PROPERTY P_Serial_fbenDTRControl : CtaSysConfig.ITF_BYTE
GET
P_Serial_fbenDTRControl := scParameter.scSerial.fbenDTRControl;
END_GET
END_PROPERTY

PROPERTY P_Serial_fbenParity : CtaSysConfig.ITF_BYTE
GET
P_Serial_fbenParity := scParameter.scSerial.fbenParity;
END_GET
END_PROPERTY

PROPERTY P_Serial_fbenRTSControl : CtaSysConfig.ITF_BYTE
GET
P_Serial_fbenRTSControl := scParameter.scSerial.fbenRTSControl;
END_GET
END_PROPERTY

PROPERTY P_Serial_fbenStopBits : CtaSysConfig.ITF_BYTE
GET
P_Serial_fbenStopBits := scParameter.scSerial.fbenStopBits;
END_GET
END_PROPERTY

PROPERTY P_Serial_fbusiNodeId : CtaSysConfig.ITF_USINT
GET
P_Serial_fbusiNodeId := scParameter.scSerial.fbusiNodeId;
END_GET
END_PROPERTY

PROPERTY P_Serial_fbxEnable : CtaSysConfig.ITF_BOOL
GET
P_Serial_fbxEnable := scParameter.scSerial.fbxEnable;
END_GET
END_PROPERTY

PROPERTY P_Serial_fbxRtuAscii : CtaSysConfig.ITF_BOOL
GET
P_Serial_fbxRtuAscii := scParameter.scSerial.fbxRtuAscii;
END_GET
END_PROPERTY

PROPERTY P_Serial_fbxEnableWatchDog : CtaSysConfig.ITF_BOOL
GET
P_Serial_fbxEnableWatchDog := scParameter.scSerial.fbxEnableWatchDog;
END_GET
END_PROPERTY

PROPERTY P_Serial_fbtWatchDog : CtaSysConfig.ITF_TIME
GET
P_Serial_fbtWatchDog := scParameter.scSerial.fbtWatchDog;
END_GET
END_PROPERTY

PROPERTY P_Serial_fbenPort : CtaSysConfig.ITF_INT
GET
P_Serial_fbenPort := scParameter.scSerial.fbenPort;
END_GET
END_PROPERTY

PROPERTY P_Tcp_fbxEnable : CtaSysConfig.ITF_BOOL
GET
P_Tcp_fbxEnable := scParameter.scTcp.fbxEnable;
END_GET
END_PROPERTY

PROPERTY P_Tcp_fbwPort : CtaSysConfig.ITF_WORD
GET
P_Tcp_fbwPort := scParameter.scTcp.fbwPort;
END_GET
END_PROPERTY

PROPERTY P_Tcp_fbxEnableWatchDog : CtaSysConfig.ITF_BOOL
GET
P_Tcp_fbxEnableWatchDog := scParameter.scTcp.fbxEnableWatchDog;
END_GET
END_PROPERTY

PROPERTY P_Tcp_fbtWatchDog : CtaSysConfig.ITF_TIME
GET
P_Tcp_fbtWatchDog := scParameter.scTcp.fbtWatchDog;
END_GET
END_PROPERTY

PROPERTY P_Tcp_fbstInterface : CtaSysConfig.ITF_STRING40
GET
P_Tcp_fbstInterface := scParameter.scTcp.fbstInterface;
END_GET
END_PROPERTY

END_FUNCTION_BLOCK

// 21 Interface/SERVER/ITF_SERVER_PARA
INTERFACE ITF_SERVER_PARA EXTENDS ITF_SERVER

PROPERTY P_Serial_fbxEnable : CtaSysConfig.ITF_BOOL
GET
END_GET
END_PROPERTY

PROPERTY P_Serial_fbusiNodeId : CtaSysConfig.ITF_USINT
GET
END_GET
END_PROPERTY

PROPERTY P_Serial_fbdwBaudrate : CtaSysConfig.ITF_DWORD
GET
END_GET
END_PROPERTY

PROPERTY P_Serial_fbbyDataBits : CtaSysConfig.ITF_BYTE
GET
END_GET
END_PROPERTY

PROPERTY P_Serial_fbenParity : CtaSysConfig.ITF_BYTE
GET
END_GET
END_PROPERTY

PROPERTY P_Serial_fbenStopBits : CtaSysConfig.ITF_BYTE
GET
END_GET
END_PROPERTY

PROPERTY P_Serial_fbenDTRControl : CtaSysConfig.ITF_BYTE
GET
END_GET
END_PROPERTY

PROPERTY P_Serial_fbenRTSControl : CtaSysConfig.ITF_BYTE
GET
END_GET
END_PROPERTY

PROPERTY P_Serial_fbxRtuAscii : CtaSysConfig.ITF_BOOL
GET
END_GET
END_PROPERTY

PROPERTY P_Serial_fbxEnableWatchDog : CtaSysConfig.ITF_BOOL
GET
END_GET
END_PROPERTY

PROPERTY P_Serial_fbtWatchDog : CtaSysConfig.ITF_TIME
GET
END_GET
END_PROPERTY

PROPERTY P_Serial_fbenPort : CtaSysConfig.ITF_INT
GET
END_GET
END_PROPERTY

PROPERTY P_Tcp_fbxEnable : CtaSysConfig.ITF_BOOL
GET
END_GET
END_PROPERTY

PROPERTY P_Tcp_fbwPort : CtaSysConfig.ITF_WORD
GET
END_GET
END_PROPERTY

PROPERTY P_Tcp_fbxEnableWatchDog : CtaSysConfig.ITF_BOOL
GET
END_GET
END_PROPERTY

PROPERTY P_Tcp_fbtWatchDog : CtaSysConfig.ITF_TIME
GET
END_GET
END_PROPERTY

PROPERTY P_Tcp_fbstInterface : CtaSysConfig.ITF_STRING40
GET
END_GET
END_PROPERTY

END_INTERFACE

// 40 Visualizations/CLIENT/CLIENT/JOBS/VIS_CLIENT_JOBS_TABLE
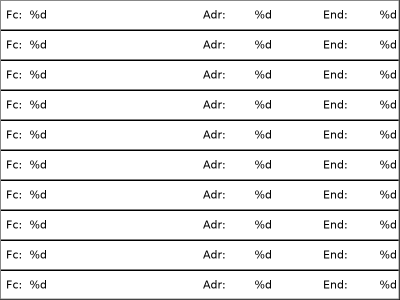
VISUALIZATION VIS_CLIENT_JOBS_TABLE  // 400x300
VAR_INPUT
	AY_ITF_MBJOB	:	ARRAY[0..9] OF ITF_MBJOB;
END_VAR
    Frame (0,0 400x30)
        shows VIS_JOB(ITF_MBJOBIN := AY_ITF_MBJOB[0])
    Frame (0,30 400x30)
        shows VIS_JOB(ITF_MBJOBIN := AY_ITF_MBJOB[1])
    Frame (0,60 400x30)
        shows VIS_JOB(ITF_MBJOBIN := AY_ITF_MBJOB[2])
    Frame (0,90 400x30)
        shows VIS_JOB(ITF_MBJOBIN := AY_ITF_MBJOB[3])
    Frame (0,120 400x30)
        shows VIS_JOB(ITF_MBJOBIN := AY_ITF_MBJOB[4])
    Frame (0,150 400x30)
        shows VIS_JOB(ITF_MBJOBIN := AY_ITF_MBJOB[5])
    Frame (0,180 400x30)
        shows VIS_JOB(ITF_MBJOBIN := AY_ITF_MBJOB[6])
    Frame (0,210 400x30)
        shows VIS_JOB(ITF_MBJOBIN := AY_ITF_MBJOB[7])
    Frame (0,240 400x30)
        shows VIS_JOB(ITF_MBJOBIN := AY_ITF_MBJOB[8])
    Frame (0,270 400x30)
        shows VIS_JOB(ITF_MBJOBIN := AY_ITF_MBJOB[9])
END_VISUALIZATION

// 40 Visualizations/CLIENT/CLIENT/JOBS/VIS_CLIENT_JOBS_QUERRY
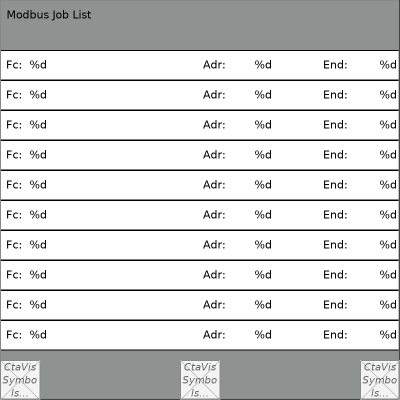
VISUALIZATION VIS_CLIENT_JOBS_QUERRY  // 400x400
VAR_INPUT
	ITF_CLIENT_IN : ITF_CLIENT;
END_VAR
    Rectangle (0,0 400x400)
    Frame (0,50 400x300)
        shows VIS_CLIENT_JOBS_TABLE(AY_ITF_MBJOB := ITF_CLIENT_IN.AY_ITF_MBJOB_VIS)
    Image (360,360 40x40), image: CtaVisSymbols.ImagePool.arrow-right_square
        OnMouseClick: execute { ITF_CLIENT_IN.RELOAD_ARRAY(FALSe,TRUE,FALSE); }
    Image (0,360 40x40), image: CtaVisSymbols.ImagePool.arrow-left_square
        OnMouseClick: execute { ITF_CLIENT_IN.RELOAD_ARRAY(FALSe,FALse,TRUE); }
    Image (180,360 40x40), image: CtaVisSymbols.ImagePool.refresh
        OnMouseClick: execute { ITF_CLIENT_IN.RELOAD_ARRAY(TRUE,FALSE,FALSE); }
    Label (0,0 200x30), "Modbus Job List"
END_VISUALIZATION

// 40 Visualizations/CLIENTMANAGER/LINE/VIS_CLIENT_LINE_QUERRY
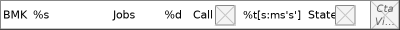
VISUALIZATION VIS_CLIENT_LINE_QUERRY  // 400x30
VAR_INPUT
	ITF_CLIENTIN		:	ITF_CLIENT;
END_VAR
    RoundedRectangle (0,0 400x30)
    Textfield (240,0 60x30), "%t[s:ms's']", text variable: ITF_CLIENTIN.ExecuteTime
    Textfield (0,0 30x30), "BMK"
    Textfield (30,0 75x30), "%s", text variable: ITF_CLIENTIN.proGetBMK
    Textfield (145,0 40x30), "%d", text variable: ITF_CLIENTIN.COUNT
    Textfield (110,0 30x30), "Jobs"
    Textfield (190,0 35x30), "Call"
    Textfield (305,0 35x30), "State"
    Image (335,5 20x20), invisible if: NOT ITF_CLIENTIN.ERROR, image: CtaVisSymbols.ImagePool.CtaError
    Image (215,5 20x20), invisible if: NOT ITF_CLIENTIN.IsCurrentCall, image: CtaVisSymbols.ImagePool.check_green
    Image (370,0 30x30), image: CtaVisSymbols.ImagePool.gear
        OnMouseClick:  Dialog=DIA_CLIENT, Parameters={ITF_CLIENT_IN: ITF_CLIENTIN}, OpenModal=True, OpenCentered=True
    Image (335,5 20x20), invisible if: ITF_CLIENTIN.ERROR, image: CtaVisSymbols.ImagePool.check_green
    RoundedRectangle (0,0 400x30)
END_VISUALIZATION

// 40 Visualizations/CLIENTMANAGER/LINE/VIS_CLIENT_LINE
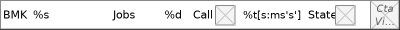
VISUALIZATION VIS_CLIENT_LINE  // 400x30
VAR_INPUT
	ITF_CLIENTIN		:	ITF_CLIENT;
END_VAR
    Frame (0,0 400x30), invisible if: NOT __QUERYINTERFACE(ITF_CLIENTIN,ITF_CLIENTIN)
        shows VIS_CLIENT_LINE_QUERRY(ITF_CLIENTIN := ITF_CLIENTIN)
END_VISUALIZATION

// 40 Visualizations/MBJOB/VIS_JOB_QUERRY
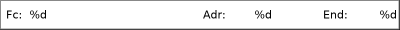
VISUALIZATION VIS_JOB_QUERRY  // 400x30
VAR_INPUT
	ITF_MBJOBIN		:	ITF_MBJOB;
END_VAR
    Rectangle (0,0 400x30)
    Textfield (0,0 25x30), "Fc:"
    Textfield (25,0 25x30), "%d", text variable: ITF_MBJOBIN.byMbFunction
    Textfield (200,0 30x30), "Adr:"
    Textfield (230,0 45x30), "%d", text variable: ITF_MBJOBIN.wMbAdress
    Textfield (320,0 30x30), "End:"
    Textfield (350,0 50x30), "%d", text variable: (ITF_MBJOBIN.wMbAdress + ITF_MBJOBIN.wQuantity-1)
    Rectangle (0,0 400x30)
END_VISUALIZATION

// 40 Visualizations/CLIENT/CLIENT/DIA_CLIENT
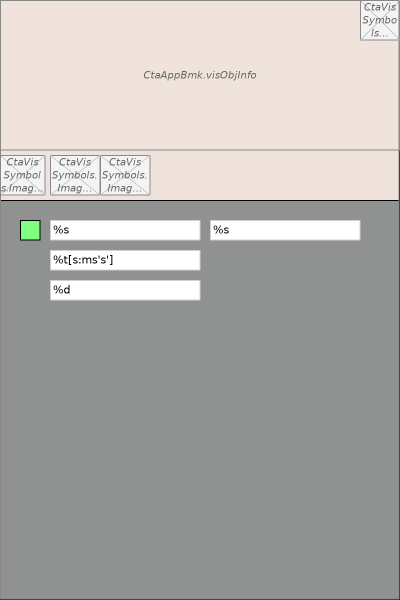
VISUALIZATION DIA_CLIENT  // 400x600
VAR_INPUT
	ITF_CLIENT_IN : ITF_CLIENT;
END_VAR
VAR
	uiPopUpGruppe 			:	UINT;
END_VAR
    Rectangle (0,0 400x600)
    Frame (0,0 400x150)
        shows CtaAppBmk.visObjInfo(ITF_BMK_IN := ITF_CLIENT_IN)
    Image (360,0 40x40), image: CtaVisSymbols.ImagePool.close_solo_black
        OnMouseClick:  Dialog=Current Dialog, Result=OK, NumpadKeypadSet=True
    Frame (0,155 400x40)
        shows VIS_CLIENT_MENÜ(uiPopUpGruppe := uiPopUpGruppe)
    Frame (0,200 400x400), frame switch variable: uiPopUpGruppe
        shows VIS_CLIENT_OVERWIEV(ITF_CLIENT_IN := ITF_CLIENT_IN)
        shows VIS_CLIENT_PARAMETER(ITF_CLIENT_IN := ITF_CLIENT_IN)
        shows VIS_CLIENT_JOBS(ITF_CLIENT_IN := ITF_CLIENT_IN)
END_VISUALIZATION

// 40 Visualizations/HELPER/VIS_IP_INPUT
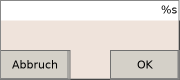
VISUALIZATION VIS_IP_INPUT  // 180x80
VAR_INPUT
    ITF_STRING40In : CtaSysConfig.ITF_STRING40;	
    stIPTemp    :   STRING;
END_VAR
    Rectangle (0,0 180x80)
    Button (110,50 70x30), "OK"
        OnMouseClick: execute {
            IF fcCheckIp(stIPTemp) THEN
                ITF_STRING40In.proValue := stIPTemp;
            ELSE
                ITF_STRING40In.proValue := 'Wrong IP';
            END_IF
        }
        OnMouseClick:  Dialog=VIS_IP_INPUT, Result=OK, NumpadKeypadSet=True
    Button (0,50 70x30), "Abbruch"
        OnMouseClick:  Dialog=VIS_IP_INPUT, Result=Cancel, NumpadKeypadSet=True
    Textfield (0,0 180x20), "%s", text variable: stIPTemp
        OnMouseClick: write the text variable via Default
END_VISUALIZATION

// 40 Visualizations/HELPER/VIS_IP_PARAMETER
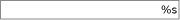
VISUALIZATION VIS_IP_PARAMETER  // 180x20
VAR_INPUT
    ITF_DATATYPE_IN : CtaSysConfig.ITF_DATATYPE;	
END_VAR
VAR
	ITF_STRING40In : CtaSysConfig.ITF_STRING40;	
END_VAR
    Frame (0,0 180x20), invisible if: NOT __QUERYINTERFACE(ITF_DATATYPE_IN,ITF_STRING40In), input disabled if: NOT __QUERYINTERFACE(ITF_DATATYPE_IN,ITF_STRING40In)
        shows VIS_IP_PARAMETER_QUERRY(ITF_STRING40In := ITF_STRING40In)
END_VISUALIZATION

// 40 Visualizations/HELPER/VIS_IP_PARAMETER_QUERRY
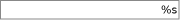
VISUALIZATION VIS_IP_PARAMETER_QUERRY  // 180x20
VAR_INPUT
    ITF_STRING40In : CtaSysConfig.ITF_STRING40;	
END_VAR
    Frame (0,0 180x20), invisible if: NOT __QUERYINTERFACE(ITF_STRING40In,ITF_STRING40In), input disabled if: NOT __QUERYINTERFACE(ITF_STRING40In,ITF_STRING40In)
        shows VIS_IP_PARAMETER_BASE(ITF_STRING40In := ITF_STRING40In)
END_VISUALIZATION

// 40 Visualizations/HELPER/VIS_IP_PARAMETER_BASE
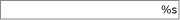
VISUALIZATION VIS_IP_PARAMETER_BASE  // 180x20
VAR_INPUT
    ITF_STRING40In : CtaSysConfig.ITF_STRING40;	
END_VAR
    Textfield (0,0 180x20), "%s", text variable: ITF_STRING40In.proValue, invisible if: NOT fcSetInitialIPString(ITF_STRING40In)
        OnMouseClick:  Dialog=VIS_IP_INPUT, Parameters={stIPTemp: ITF_STRING40In.proValue, ITF_STRING40In: ITF_STRING40In}, OpenModal=True, OpenCentered=True
END_VISUALIZATION

// 40 Visualizations/MBJOB/VIS_JOB
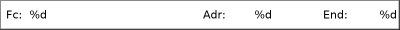
VISUALIZATION VIS_JOB  // 400x30
VAR_INPUT
	ITF_MBJOBIN		:	ITF_MBJOB;
END_VAR
    Frame (0,0 400x30), invisible if: NOT __QUERYINTERFACE(ITF_MBJOBIN,ITF_MBJOBIN)
        shows VIS_JOB_QUERRY(ITF_MBJOBIN := ITF_MBJOBIN)
END_VISUALIZATION

// 40 Visualizations/CLIENTMANAGER/MENÜ/VIS_CLIENTMANAGER_MENÜ
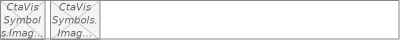
VISUALIZATION VIS_CLIENTMANAGER_MENÜ  // 400x40
VAR_IN_OUT
	uiPopUpGruppe 			:	UINT;
END_VAR
    Rectangle (50,0 40x40), colour toggle: uiPopUpGruppe = 1
        OnMouseDown: execute { uiPopUpGruppe := 1; }
    Rectangle (0,0 40x40), colour toggle: uiPopUpGruppe = 0
        OnMouseDown: execute { uiPopUpGruppe := 0; }
    Image (0,0 45x40), image: CtaVisSymbols.ImagePool.eye
        OnMouseDown: execute { uiPopUpGruppe := 0; }
    Image (50,0 50x40), image: CtaVisSymbols.ImagePool.gear
        OnMouseDown: execute { uiPopUpGruppe := 1; }
END_VISUALIZATION

// 40 Visualizations/CLIENTMANAGER/DIA_CLIENT_MANAGER
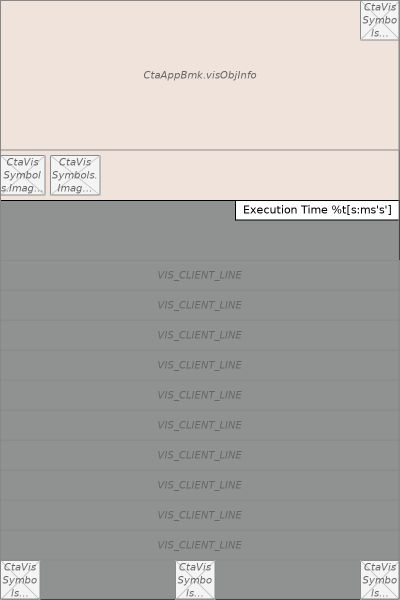
VISUALIZATION DIA_CLIENT_MANAGER  // 400x600
VAR_INPUT
	ITF_CLIENT_MANAGER_IN : ITF_MB_CLIENTMANAGER;
END_VAR
VAR
	uiPopUpGruppe 			:	UINT;
END_VAR
    Rectangle (0,0 400x600)
    Frame (0,200 400x400), invisible if: NOT __QUERYINTERFACE(ITF_CLIENT_MANAGER_IN,ITF_CLIENT_MANAGER_IN), frame switch variable: uiPopUpGruppe
        shows VIS_CLIENT_MANAGER_OVERWIEV(ITF_CLIENT_MANAGER_IN := ITF_CLIENT_MANAGER_IN)
        shows VIS_CLIENT_MANAGER_PARAMETER(ITF_CLIENT_MANAGER_IN := ITF_CLIENT_MANAGER_IN)
    Image (360,0 40x40), image: CtaVisSymbols.ImagePool.close_solo_black
        OnMouseClick:  Dialog=Current Dialog, Result=OK, NumpadKeypadSet=True
    Frame (0,155 400x40)
        shows VIS_CLIENTMANAGER_MENÜ(uiPopUpGruppe := uiPopUpGruppe)
    Frame (0,0 400x150)
        shows CtaAppBmk.visObjInfo()
END_VISUALIZATION

// 40 Visualizations/CLIENTMANAGER/OVERWIEV/VIS_CLIENT_MANAGER_OVERWIEV_QUERRY
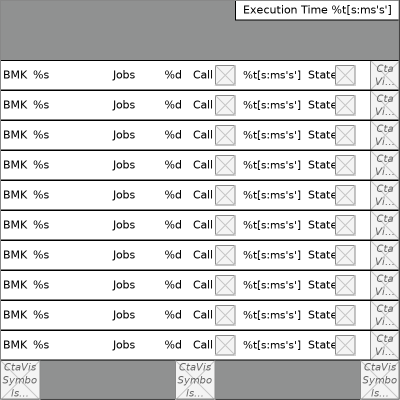
VISUALIZATION VIS_CLIENT_MANAGER_OVERWIEV_QUERRY  // 400x400
VAR_INPUT
	ITF_CLIENT_MANAGER_IN : ITF_MB_CLIENTMANAGER;
END_VAR
    Rectangle (0,0 400x400)
    Image (360,360 40x40), image: CtaVisSymbols.ImagePool.arrow-right_square
        OnMouseClick: execute { ITF_CLIENT_MANAGER_IN.RELOAD_ARRAY(FALSe,TRUE,FALSE); }
    Image (0,360 40x40), image: CtaVisSymbols.ImagePool.arrow-left_square
        OnMouseClick: execute { ITF_CLIENT_MANAGER_IN.RELOAD_ARRAY(FALSe,FALse,TRUE); }
    Image (175,360 40x40), image: CtaVisSymbols.ImagePool.refresh
        OnMouseClick: execute { ITF_CLIENT_MANAGER_IN.RELOAD_ARRAY(TRUE,FALSE,FALSE); }
    Textfield (235,0 165x20), "Execution Time %t[s:ms's']", text variable: ITF_CLIENT_MANAGER_IN.OperationTime
    Frame (0,60 400x300)
        shows VIS_CLIENT_MANAGER_TABLE(AY_ITF_CLIENTS := ITF_CLIENT_MANAGER_IN.AY_ITF_MBCLIENT_VIS)
END_VISUALIZATION

// 40 Visualizations/CLIENTMANAGER/OVERWIEV/VIS_CLIENT_MANAGER_TABLE
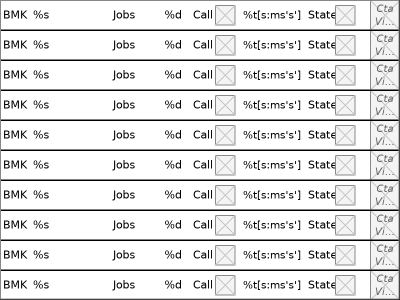
VISUALIZATION VIS_CLIENT_MANAGER_TABLE  // 400x300
VAR_INPUT
	AY_ITF_CLIENTS	:	ARRAY[0..9] OF ITF_CLIENT;
END_VAR
    Frame (0,0 400x30)
        shows VIS_CLIENT_LINE(ITF_CLIENTIN := AY_ITF_CLIENTS[0])
    Frame (0,30 400x30)
        shows VIS_CLIENT_LINE(ITF_CLIENTIN := AY_ITF_CLIENTS[1])
    Frame (0,60 400x30)
        shows VIS_CLIENT_LINE(ITF_CLIENTIN := AY_ITF_CLIENTS[2])
    Frame (0,90 400x30)
        shows VIS_CLIENT_LINE(ITF_CLIENTIN := AY_ITF_CLIENTS[3])
    Frame (0,120 400x30)
        shows VIS_CLIENT_LINE(ITF_CLIENTIN := AY_ITF_CLIENTS[4])
    Frame (0,150 400x30)
        shows VIS_CLIENT_LINE(ITF_CLIENTIN := AY_ITF_CLIENTS[5])
    Frame (0,180 400x30)
        shows VIS_CLIENT_LINE(ITF_CLIENTIN := AY_ITF_CLIENTS[6])
    Frame (0,210 400x30)
        shows VIS_CLIENT_LINE(ITF_CLIENTIN := AY_ITF_CLIENTS[7])
    Frame (0,240 400x30)
        shows VIS_CLIENT_LINE(ITF_CLIENTIN := AY_ITF_CLIENTS[8])
    Frame (0,270 400x30)
        shows VIS_CLIENT_LINE(ITF_CLIENTIN := AY_ITF_CLIENTS[9])
END_VISUALIZATION

// 40 Visualizations/CLIENT/CLIENT/MENÜ/VIS_CLIENT_MENÜ
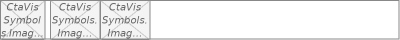
VISUALIZATION VIS_CLIENT_MENÜ  // 400x40
VAR_IN_OUT
	uiPopUpGruppe 			:	UINT;
END_VAR
    Rectangle (100,0 40x40), colour toggle: uiPopUpGruppe = 2
        OnMouseDown: execute { uiPopUpGruppe := 2; }
    Rectangle (50,0 40x40), colour toggle: uiPopUpGruppe = 1
        OnMouseDown: execute { uiPopUpGruppe := 1; }
    Rectangle (0,0 40x40), colour toggle: uiPopUpGruppe = 0
        OnMouseDown: execute { uiPopUpGruppe := 0; }
    Image (0,0 45x40), image: CtaVisSymbols.ImagePool.eye
        OnMouseDown: execute { uiPopUpGruppe := 0; }
    Image (50,0 50x40), image: CtaVisSymbols.ImagePool.gear
        OnMouseDown: execute { uiPopUpGruppe := 1; }
    Image (100,0 50x40), image: CtaVisSymbols.ImagePool.lan
        OnMouseDown: execute { uiPopUpGruppe := 2; }
END_VISUALIZATION

// 40 Visualizations/CLIENT/CLIENT/OVERWIEV/VIS_CLIENT_OVERWIEV
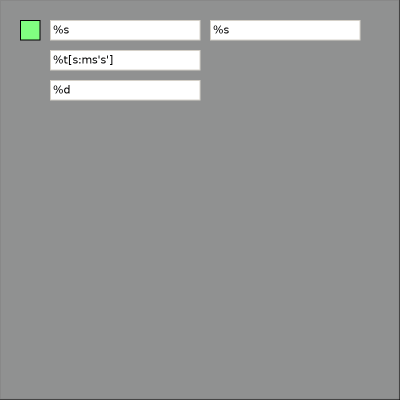
VISUALIZATION VIS_CLIENT_OVERWIEV  // 400x400
VAR_INPUT
	ITF_CLIENT_IN : ITF_CLIENT;	
END_VAR
    Frame (0,0 400x400), invisible if: NOT __QUERYINTERFACE(ITF_CLIENT_IN,ITF_CLIENT_IN)
        shows VIS_CLIENT_OVERWIEV_QUERY(ITF_CLIENT_IN := ITF_CLIENT_IN)
END_VISUALIZATION

// 40 Visualizations/CLIENT/CLIENT/PARAMETER/VIS_CLIENT_PARAMETER
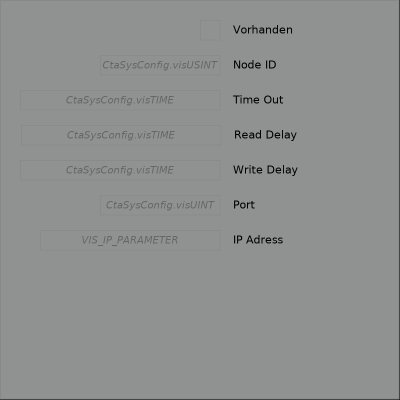
VISUALIZATION VIS_CLIENT_PARAMETER  // 400x400
VAR_INPUT
	ITF_CLIENT_IN : ITF_CLIENT;	
END_VAR
    Rectangle (0,0 400x400)
    Frame (0,0 400x400)
        shows VIS_CLIENT_PARAMETER_RTU(ITF_CLIENT_IN := ITF_CLIENT_IN)
    Frame (0,0 400x400)
        shows VIS_CLIENT_PARAMETER_TCP(ITF_CLIENT_IN := ITF_CLIENT_IN)
END_VISUALIZATION

// 40 Visualizations/CLIENT/CLIENT/OVERWIEV/VIS_CLIENT_OVERWIEV_QUERY
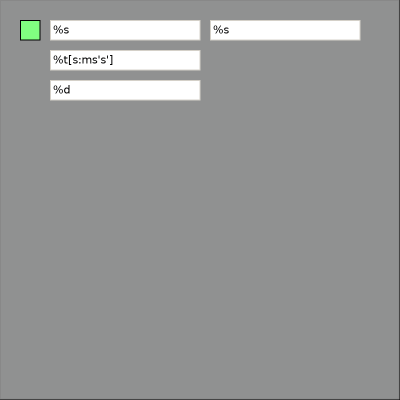
VISUALIZATION VIS_CLIENT_OVERWIEV_QUERY  // 400x400
VAR_INPUT
	ITF_CLIENT_IN : ITF_CLIENT;	
END_VAR
    Rectangle (0,0 400x400)
    Rectangle (20,20 20x20), colour toggle: ITF_CLIENT_IN.ERROR
    Textfield (50,20 150x20), "%s", text variable: TO_STRING(ITF_CLIENT_IN.ERROR_ID)
    Textfield (210,20 150x20), "%s", text variable: TO_STRING(ITF_CLIENT_IN.EXEPTION_CODE)
    Textfield (50,50 150x20), "%t[s:ms's']", text variable: ITF_CLIENT_IN.ExecuteTime
    Textfield (50,80 150x20), "%d", text variable: ITF_CLIENT_IN.COUNT
END_VISUALIZATION

// 40 Visualizations/CLIENT/CLIENT/JOBS/VIS_CLIENT_JOBS
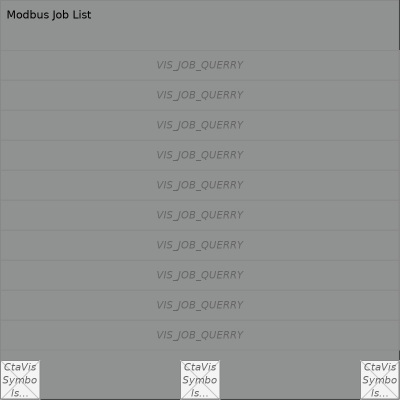
VISUALIZATION VIS_CLIENT_JOBS  // 400x400
VAR_INPUT
	ITF_CLIENT_IN : ITF_CLIENT;	
END_VAR
    Frame (0,0 400x400), invisible if: NOT __QUERYINTERFACE(ITF_CLIENT_IN,ITF_CLIENT_IN)
        shows VIS_CLIENT_JOBS_QUERRY(ITF_CLIENT_IN := ITF_CLIENT_IN)
END_VISUALIZATION

// 40 Visualizations/CLIENT/RTU/PARAMETER/VIS_CLIENT_PARAMETER_RTU
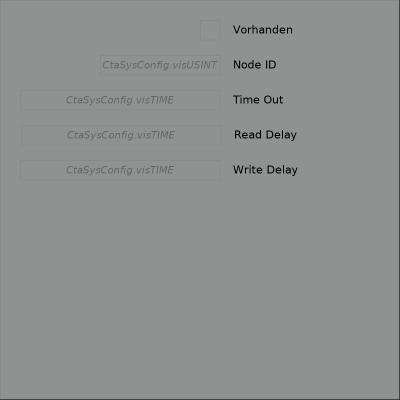
VISUALIZATION VIS_CLIENT_PARAMETER_RTU  // 400x400
VAR_INPUT
	ITF_CLIENT_IN : ITF_CLIENT;	
END_VAR
VAR
	ITF_MB_CLIENT_RTU_QUERY	:	ITF_MB_CLIENT_RTU;
END_VAR
    Frame (0,0 400x400), invisible if: NOT __QUERYINTERFACE(ITF_CLIENT_IN,ITF_MB_CLIENT_RTU_QUERY)
        shows VIS_CLIENT_PARAMETER_RTU_TEMP(ITF_MB_CLIENT_RTU_QUERY := ITF_MB_CLIENT_RTU_QUERY)
END_VISUALIZATION

// 40 Visualizations/CLIENT/RTU/PARAMETER/VIS_CLIENT_PARAMETER_RTU_QUERY
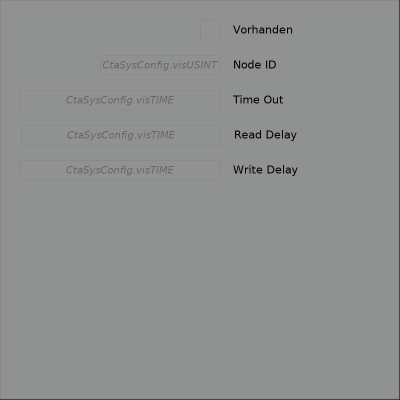
VISUALIZATION VIS_CLIENT_PARAMETER_RTU_QUERY  // 400x400
VAR_INPUT
	ITF_MB_CLIENT_RTU_IN : ITF_MB_CLIENT_RTU;	
END_VAR
    Rectangle (0,0 400x400)
    Frame (200,20 20x20)
        shows CtaSysConfig.visBOOL(visfbBOOLIn := ITF_MB_CLIENT_RTU_IN.P_fbxEnable)
    Label (230,20 150x20), "Vorhanden"
    Label (230,55 150x20), "Node ID"
    Frame (100,55 120x20)
        shows CtaSysConfig.visUSINT(visfbUSINTIn := ITF_MB_CLIENT_RTU_IN.P_fbusiNodeId)
    Label (230,90 150x20), "Time Out"
    Frame (20,90 200x20)
        shows CtaSysConfig.visTIME(visfbTIMEIn := ITF_MB_CLIENT_RTU_IN.P_fbtTimeOut)
    Frame (21,125 200x20)
        shows CtaSysConfig.visTIME(visfbTIMEIn := ITF_MB_CLIENT_RTU_IN.P_fbtReadDelay)
    Label (231,125 150x20), "Read Delay"
    Frame (20,160 200x20)
        shows CtaSysConfig.visTIME(visfbTIMEIn := ITF_MB_CLIENT_RTU_IN.P_fbtWriteDelay)
    Label (230,160 150x20), "Write Delay"
END_VISUALIZATION

// 40 Visualizations/CLIENT/TCP/PARAMETER/VIS_CLIENT_PARAMETER_TCP
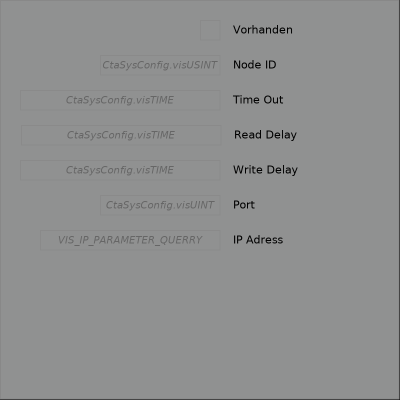
VISUALIZATION VIS_CLIENT_PARAMETER_TCP  // 400x400
VAR_INPUT
	ITF_CLIENT_IN : ITF_CLIENT;	
END_VAR
VAR
	ITF_MB_CLIENT_TCP_QUERY	:	ITF_MB_CLIENT_TCP;
END_VAR
    Frame (0,0 400x400), invisible if: NOT __QUERYINTERFACE(ITF_CLIENT_IN,ITF_MB_CLIENT_TCP_QUERY)
        shows VIS_CLIENT_PARAMETER_TCP_TEMP(ITF_MB_CLIENT_TCP_QUERY := ITF_MB_CLIENT_TCP_QUERY)
END_VISUALIZATION

// 40 Visualizations/CLIENT/TCP/PARAMETER/VIS_CLIENT_PARAMETER_TCP_QUERY
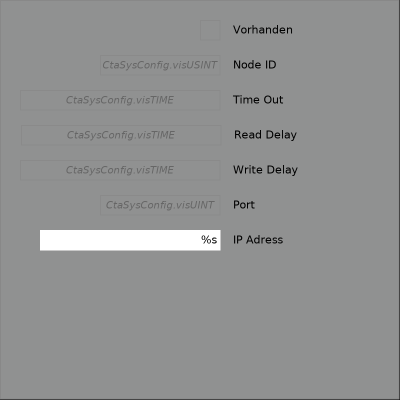
VISUALIZATION VIS_CLIENT_PARAMETER_TCP_QUERY  // 400x400
VAR_INPUT
	ITF_MB_CLIENT_TCP_IN : ITF_MB_CLIENT_TCP;	
END_VAR
    Rectangle (0,0 400x400)
    Frame (200,20 20x20)
        shows CtaSysConfig.visBOOL(visfbBOOLIn := ITF_MB_CLIENT_TCP_IN.P_fbxEnable)
    Label (230,20 150x20), "Vorhanden"
    Label (230,55 150x20), "Node ID"
    Frame (100,55 120x20)
        shows CtaSysConfig.visUSINT(visfbUSINTIn := ITF_MB_CLIENT_TCP_IN.P_fbusiNodeId)
    Label (230,90 150x20), "Time Out"
    Frame (20,90 200x20)
        shows CtaSysConfig.visTIME(visfbTIMEIn := ITF_MB_CLIENT_TCP_IN.P_fbtTimeOut)
    Frame (21,125 200x20)
        shows CtaSysConfig.visTIME(visfbTIMEIn := ITF_MB_CLIENT_TCP_IN.P_fbtReadDelay)
    Label (231,125 150x20), "Read Delay"
    Frame (20,160 200x20)
        shows CtaSysConfig.visTIME(visfbTIMEIn := ITF_MB_CLIENT_TCP_IN.P_fbtWriteDelay)
    Label (230,160 150x20), "Write Delay"
    Label (230,195 150x20), "Port"
    Frame (100,195 120x20)
        shows CtaSysConfig.visUINT(visfbUINTIn := ITF_MB_CLIENT_TCP_IN.P_fbuiPort)
    Label (230,230 150x20), "IP Adress"
    Frame (40,230 180x20)
        shows VIS_IP_PARAMETER(ITF_DATATYPE_IN := ITF_MB_CLIENT_TCP_IN.P_fbstIpAdress)
END_VISUALIZATION

// 40 Visualizations/CLIENTMANAGER/PARAMETER/VIS_CLIENT_MANAGER_PARAMETER
